TYPE ST_Event :
STRUCT
	eEventType : E_EventType; //user defined ENUM
	eEventSeverity : TcEventSeverity; // library ENUM
	nEventIdentity : UDINT;
	sEvenText : STRING(255);
	dtTimestamp : DATE_AND_TIME;
END_STRUCT
END_TYPE

(* stored: Version 1.1.0.1, ProductVersion 3.1.4024.10
   DUT ST_Event: Id {8dd7bb5d-b643-4621-b685-f59effc9d0c8} *)
